FUNCTION_BLOCK FirstState IMPLEMENTS Istate
VAR
	stateFinished: BOOL;
	_description: STRING := 'FirstState';
END_VAR

PROPERTY Description : STRING
GET
Description:= _description;
END_GET
END_PROPERTY

METHOD execute : BOOL
IF NOT stateFinished THEN 
	THIS^();
END_IF

execute:= stateFinished;
END_METHOD

///FB_Init is always available implicitly and it is used primarily for initialization.
///The return value is not evaluated. For a specific influence, you can also declare the
///methods explicitly and provide additional code there with the standard initialization
///code. You can evaluate the return value.
METHOD FB_Init : BOOL
VAR_INPUT
	/// TRUE: the retain variables are initialized (reset warm / reset cold)
	bInitRetains: BOOL;
	/// TRUE: the instance will be copied to the copy code afterward (online change) 
	bInCopyCode: BOOL;
END_VAR
END_METHOD

END_FUNCTION_BLOCK

(* stored: Version 1.1.0.1
   POU FirstState: Id {e8dc026b-c3a1-48fd-af49-4305811eb2f1}, SpecialFunc None
   Property Description: Id {9daa34d6-2636-4c68-acff-8d0f5563ccaf}
   Get Get: Id {001f5a43-3d7a-45b1-b3a0-60aa26f73884}
   Method execute: Id {393d3478-e1f6-47da-ad24-b3df47e6be45}
   Method FB_Init: Id {b20b5e01-02df-4dcf-8611-514c6ad0941f} *)
